// TIA Portal V19 export
FUNCTION_BLOCK "GRAFCET"   // FB1, GRAPH
   VAR_INPUT
      OFF_SQ { ExternalAccessible := 'False'; ExternalVisible := 'False'; ExternalWritable := 'False'} : Bool := false;   // Turn sequence off
      INIT_SQ { ExternalAccessible := 'False'; ExternalVisible := 'False'; ExternalWritable := 'False'} : Bool := false;   // Set sequence to initial state
      ACK_EF { ExternalAccessible := 'False'; ExternalVisible := 'False'; ExternalWritable := 'False'} : Bool := false;   // Acknowledge all errors and faults
      S_PREV { ExternalAccessible := 'False'; ExternalVisible := 'False'; ExternalWritable := 'False'} : Bool := false;   // Output previous step in parameter S_NO
      S_NEXT { ExternalAccessible := 'False'; ExternalVisible := 'False'; ExternalWritable := 'False'} : Bool := false;   // Indicate next step in parameter S_NO
      SW_AUTO { ExternalAccessible := 'False'; ExternalVisible := 'False'; ExternalWritable := 'False'} : Bool := false;   // Automatic mode
      SW_TAP { ExternalAccessible := 'False'; ExternalVisible := 'False'; ExternalWritable := 'False'} : Bool := false;   // Semiautomatic/switch with transition
      SW_TOP { ExternalAccessible := 'False'; ExternalVisible := 'False'; ExternalWritable := 'False'} : Bool := false;   // Semiautomatic/ignore transition
      SW_MAN { ExternalAccessible := 'False'; ExternalVisible := 'False'; ExternalWritable := 'False'} : Bool := false;   // Manual mode
      S_SEL { ExternalAccessible := 'False'; ExternalVisible := 'False'; ExternalWritable := 'False'} : Int := 0;   // Select step to be output to S_NO
      S_ON { ExternalAccessible := 'False'; ExternalVisible := 'False'; ExternalWritable := 'False'} : Bool := false;   // Activate step indicated in S_NO
      S_OFF { ExternalAccessible := 'False'; ExternalVisible := 'False'; ExternalWritable := 'False'} : Bool := false;   // Deactivate step indicated S_NO
      T_PUSH { ExternalAccessible := 'False'; ExternalVisible := 'False'; ExternalWritable := 'False'} : Bool := false;   // Enable transition to switch in semi automatic mode
   END_VAR
   VAR_OUTPUT
      S_NO { ExternalAccessible := 'False'; ExternalVisible := 'False'; ExternalWritable := 'False'} : Int := 0;   // Step number
      S_MORE { ExternalAccessible := 'False'; ExternalVisible := 'False'; ExternalWritable := 'False'} : Bool := false;   // More steps are available and can be shown in S_NO
      S_ACTIVE { ExternalAccessible := 'False'; ExternalVisible := 'False'; ExternalWritable := 'False'} : Bool := false;   // Step indicated in S_NO is active
      ERR_FLT { ExternalAccessible := 'False'; ExternalVisible := 'False'; ExternalWritable := 'False'} : Bool := false;   // Interlock or supervision group error
      AUTO_ON { ExternalAccessible := 'False'; ExternalVisible := 'False'; ExternalWritable := 'False'} : Bool := false;   // Automatic mode is active
      TAP_ON { ExternalAccessible := 'False'; ExternalVisible := 'False'; ExternalWritable := 'False'} : Bool := false;   // Semiautomatic mode/step with transition enabled
      TOP_ON { ExternalAccessible := 'False'; ExternalVisible := 'False'; ExternalWritable := 'False'} : Bool := false;   // Semiautomatic mode/ignore transition enabled
      MAN_ON { ExternalAccessible := 'False'; ExternalVisible := 'False'; ExternalWritable := 'False'} : Bool := false;   // Manual mode is active
   END_VAR
   VAR
      S_DISPLAY { ExternalAccessible := 'False'; ExternalVisible := 'False'; ExternalWritable := 'False'} : Int;   // Internal display of output parameter S_NO
      S_SEL_OLD { ExternalAccessible := 'False'; ExternalVisible := 'False'; ExternalWritable := 'False'} : Int;   // Previous value in S_SEL
      S_DISPIDX { ExternalAccessible := 'False'; ExternalVisible := 'False'; ExternalWritable := 'False'} : Byte;   // Index of the step in S_NO
      T_DISPIDX { ExternalAccessible := 'False'; ExternalVisible := 'False'; ExternalWritable := 'False'} : Byte;   // Index of the transition displayed in T_NO
      MOP { ExternalAccessible := 'False'; ExternalVisible := 'False'; ExternalWritable := 'False'} : Struct   // Mode
         AUTO : Bool := true;   // Status: automatic mode
         MAN : Bool := false;   // Status: manual mode
         TAP : Bool := false;   // Status: semi automatic/switch with transition
         TOP : Bool := false;   // Status: semi automatic/ignore transition
         ACK_S : Bool := false;   // Request: acknowledge step at parameter S_NO
         REG_S : Bool := false;   // Request: register step indicated in S_NO
         T_PREV : Bool := false;   // Request: output previous valid transition in T_NO
         T_NEXT : Bool := false;   // Request: output next valid transition in T_NO
         LOCK : Bool := true;   // Status: interlocks activated
         SUP : Bool := true;   // Status: supervisions activated
         ACKREQ : Bool := true;   // Status: acknowledgment required
         SSKIP : Bool := false;   // Status: "Skip steps" enabled
         OFF : Bool := false;   // Request: deactivate all steps
         INIT : Bool := true;   // Request: set sequence to initial state
         HALT : Bool := false;   // Status: sequence halted
         TMS_HALT : Bool := false;   // Status: all internal timers held
         OPS_ZERO : Bool := false;   // Status: set all operands processed with N, L, D instructions to 0
         SACT_DISP : Bool := true;   // Status: display active steps only
         SEF_DISP : Bool := false;   // Status: display only steps with errors and disrupted steps
         SALL_DISP : Bool := false;   // Status: display all steps
         S_PREV : Bool := false;   // Request: output previous step to S_NO
         S_NEXT : Bool := false;   // Request: Output next step at S_NO parameter
         S_SELOK : Bool := false;   // Request: output step number from S_SEL to S_NO
         S_ON : Bool := false;   // Request: activate step indicated in S_NO
         S_OFF : Bool := false;   // Request: deactivate step at parameter S_NO
         T_PUSH : Bool := false;   // Request: transition switching enabled
         REG : Bool := false;   // Request: register all interlock and supervision errors
         ACK : Bool := false;   // Request: acknowledge all interlock and supervision errors
         IL_PERM : Bool := false;   // Status: permanent processing of all interlocks
         T_PERM : Bool := false;   // Status: permanent processing of all transitions
         ILP_MAN : Bool := false;   // Status: permanent processing of all interlocks in manual mode
      END_STRUCT;
      TICKS { ExternalAccessible := 'False'; ExternalVisible := 'False'; ExternalWritable := 'False'} : Struct   // Clock speeds
         DELTA : Time := T#0ms;   // Time difference between cycles
         OLD : Time := T#0ms;   // 10 ms clock counter value in last cycle
         NEW : Time := T#0ms;   // 10 ms clock counter value in this cycle
      END_STRUCT;
      SQ_FLAGS { ExternalAccessible := 'False'; ExternalVisible := 'False'; ExternalWritable := 'False'} : Struct   // Sequence bit memory
         ERR_FLT : Bool := false;   // Interlock and supervision group error
         ERROR : Bool := false;   // Interlock group error
         FAULT : Bool := false;   // Supervision group error
         RT_FAIL : Bool := false;   // Runtime error
         NO_SNO : Bool := false;   // Requested step number not found
         NF_OFL : Bool := false;   // Overflow: too many ON or OFF requests
         SA_OFL : Bool := false;   // Overflow: too many steps active
         TV_OFL : Bool := false;   // Overflow: too many valid transitions
         MSG_OFL : Bool := false;   // Overflow: not enough system resources for ALARM_S
         NO_SWI : Bool := false;   // Do not switch in this cycle
         CYC_OP : Bool := false;   // Cyclic execution of the sequence after initialization
         AS_MSG : Bool := true;   // Alarms during runtime enabled or disabled by instruction
         AS_SEND : Bool := false;   // Send alarms from WR_USMSG or only enter in diagnostics buffer
         SQ_BUSY : Bool := false;   // Internal edge bit memory for sequence processing
         SA_BUSY : Bool := false;   // Internal edge bit memory for sequence processing
         AS_SIG : Bool := false;   // Edge bit memory for alarms from Alarm_S and Alarm_SQ
      END_STRUCT;
   END_VAR
BEGIN
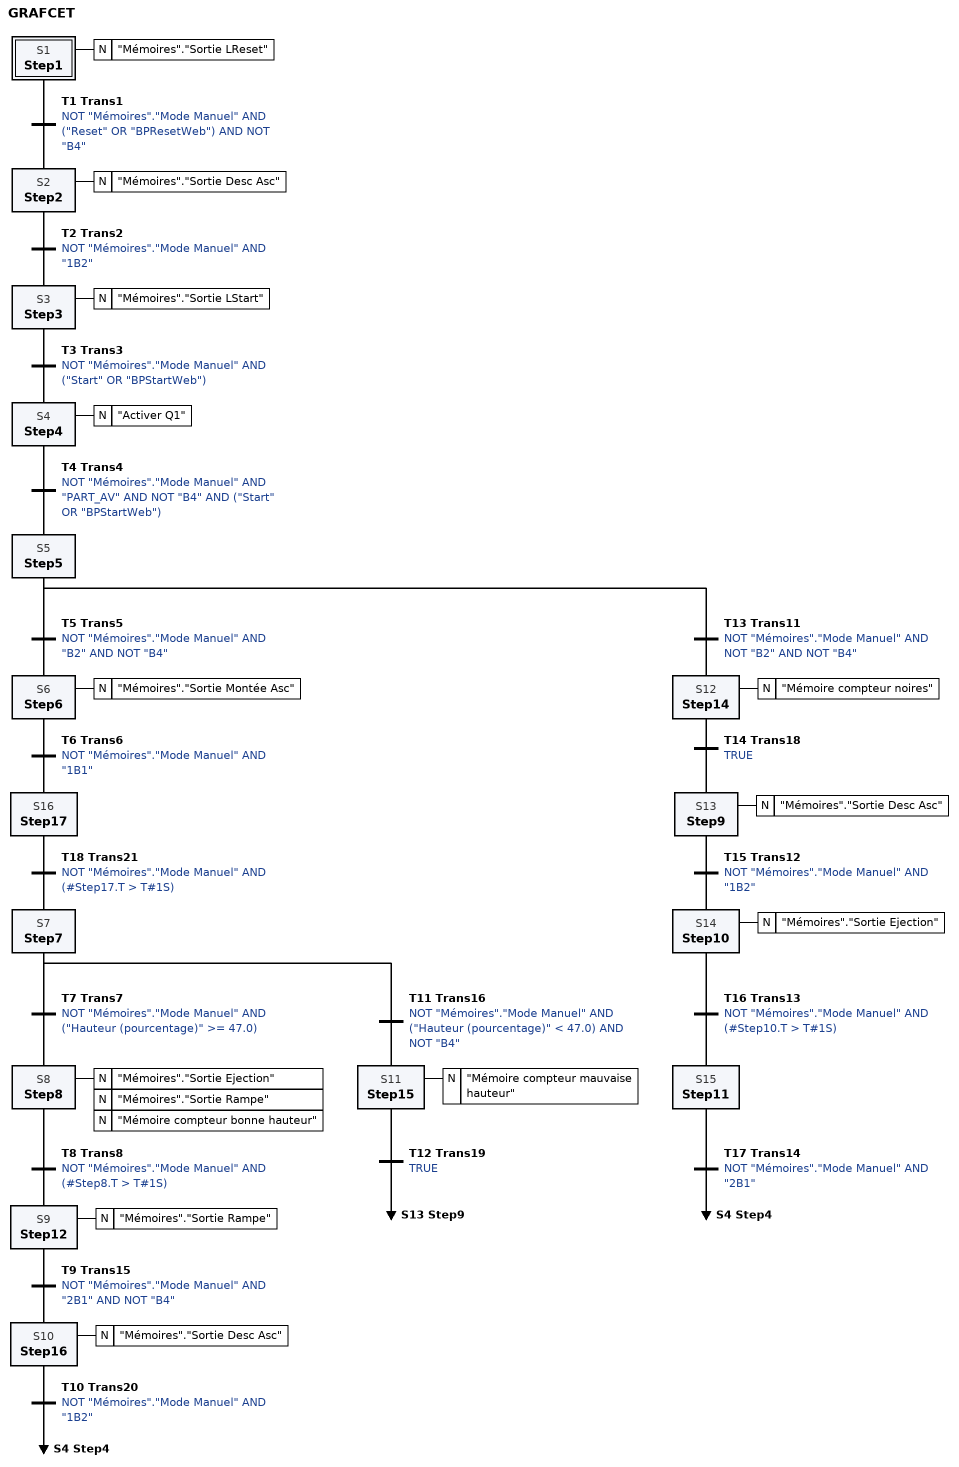
   // sequencer 1: GRAFCET de la séquence de tri
   INITIAL_STEP Step1:   // S1
              N    "Mémoires"."Sortie LReset"
   END_STEP
   TRANSITION Trans1 FROM Step1 TO Step2   // T1
      := NOT "Mémoires"."Mode Manuel" AND ("Reset" OR "BPResetWeb") AND NOT "B4";
   END_TRANSITION
   STEP Step2:   // S2
              N    "Mémoires"."Sortie Desc Asc"
   END_STEP
   TRANSITION Trans2 FROM Step2 TO Step3   // T2
      := NOT "Mémoires"."Mode Manuel" AND "1B2";
   END_TRANSITION
   STEP Step3:   // S3
              N    "Mémoires"."Sortie LStart"
   END_STEP
   TRANSITION Trans3 FROM Step3 TO Step4   // T3
      := NOT "Mémoires"."Mode Manuel" AND ("Start" OR "BPStartWeb");
   END_TRANSITION
   STEP Step4:   // S4
              N    "Activer Q1"
   END_STEP
   TRANSITION Trans4 FROM Step4 TO Step5   // T4
      := NOT "Mémoires"."Mode Manuel" AND "PART_AV" AND NOT "B4" AND ("Start" OR "BPStartWeb");
   END_TRANSITION
   STEP Step5:   // S5
   END_STEP
   TRANSITION Trans5 FROM Step5 TO Step6   // T5
      := NOT "Mémoires"."Mode Manuel" AND "B2" AND NOT "B4";
   END_TRANSITION
   TRANSITION Trans11 FROM Step5 TO Step14   // T13
      := NOT "Mémoires"."Mode Manuel" AND NOT "B2" AND NOT "B4";
   END_TRANSITION
   STEP Step6:   // S6
              N    "Mémoires"."Sortie Montée Asc"
   END_STEP
   TRANSITION Trans6 FROM Step6 TO Step17   // T6
      := NOT "Mémoires"."Mode Manuel" AND "1B1";
   END_TRANSITION
   STEP Step7:   // S7
   END_STEP
   TRANSITION Trans7 FROM Step7 TO Step8   // T7
      := NOT "Mémoires"."Mode Manuel" AND ("Hauteur (pourcentage)" >= 47.0);
   END_TRANSITION
   TRANSITION Trans16 FROM Step7 TO Step15   // T11
      := NOT "Mémoires"."Mode Manuel" AND ("Hauteur (pourcentage)" < 47.0) AND NOT "B4";
   END_TRANSITION
   STEP Step8:   // S8
              N    "Mémoires"."Sortie Ejection"
              N    "Mémoires"."Sortie Rampe"
              N    "Mémoire compteur bonne hauteur"
   END_STEP
   TRANSITION Trans8 FROM Step8 TO Step12   // T8
      := NOT "Mémoires"."Mode Manuel" AND (#Step8.T > T#1S);
   END_TRANSITION
   STEP Step9:   // S13
              N    "Mémoires"."Sortie Desc Asc"
   END_STEP
   TRANSITION Trans12 FROM Step9 TO Step10   // T15
      := NOT "Mémoires"."Mode Manuel" AND "1B2";
   END_TRANSITION
   STEP Step10:   // S14
              N    "Mémoires"."Sortie Ejection"
   END_STEP
   TRANSITION Trans13 FROM Step10 TO Step11   // T16
      := NOT "Mémoires"."Mode Manuel" AND (#Step10.T > T#1S);
   END_TRANSITION
   STEP Step11:   // S15
   END_STEP
   TRANSITION Trans14 FROM Step11 TO Step4   // T17, jump
      := NOT "Mémoires"."Mode Manuel" AND "2B1";
   END_TRANSITION
   STEP Step12:   // S9
              N    "Mémoires"."Sortie Rampe"
   END_STEP
   TRANSITION Trans15 FROM Step12 TO Step16   // T9
      := NOT "Mémoires"."Mode Manuel" AND "2B1" AND NOT "B4";
   END_TRANSITION
   STEP Step14:   // S12
              N    "Mémoire compteur noires"
   END_STEP
   TRANSITION Trans18 FROM Step14 TO Step9   // T14
      := TRUE;
   END_TRANSITION
   STEP Step15:   // S11
              N    "Mémoire compteur mauvaise hauteur"
   END_STEP
   TRANSITION Trans19 FROM Step15 TO Step9   // T12, jump
      := TRUE;
   END_TRANSITION
   STEP Step16:   // S10
              N    "Mémoires"."Sortie Desc Asc"
   END_STEP
   TRANSITION Trans20 FROM Step16 TO Step4   // T10, jump
      := NOT "Mémoires"."Mode Manuel" AND "1B2";
   END_TRANSITION
   STEP Step17:   // S16
   END_STEP
   TRANSITION Trans21 FROM Step17 TO Step7   // T18
      := NOT "Mémoires"."Mode Manuel" AND (#Step17.T > T#1S);
   END_TRANSITION
END_FUNCTION_BLOCK
